TYPE ST_BA_BuildingAlarms :
STRUCT
	bBurglary				: BOOL;
	bFireAlert				: BOOL;
	bCentralOff				: BOOL;
	bForcedVentilation		: BOOL;
	bSmokeExtraction		: BOOL;
END_STRUCT
END_TYPE

(* stored: Version 1.1.0.1, ProductVersion 3.1.4024.6
   DUT ST_BA_BuildingAlarms: Id {c2475f00-ac04-4b26-b72b-5f0a66736357} *)
